VAR_GLOBAL
	HmiToPlc	: ARRAY[1..MAX_AXES] OF Motion_HmiToPlc;
	PlcToHmi	: ARRAY[1..MAX_AXES] OF Motion_PlcToHmi;
	AXIS		: ARRAY[1..MAX_AXES] OF Motion_Axis;
END_VAR

(* stored: Version 1.1.0.1, ProductVersion 3.1.0.36
   GVL ServoMotion_GVL: Id {72aa564a-0c5e-4f07-995d-938fcc730134} *)
